// TIA Portal project "SortowanieNiebieskiZielony" (V17)
// Vorlageprojekt für das Buch mit Zielsystem S7-1200

(* hardware
DEVICE "S7-1200-Station_1"  S7-1200 Station
   slot 0: "Baugruppenträger_0"  Rack  V1.0
   slot 1: "PLC_1"  CPU 1211C DC/DC/DC  6ES7 211-1AE40-0XB0  V4.1
*)

// ===== PLC "PLC_1"  CPU 1211C DC/DC/DC =====

VAR_GLOBAL   // PLC tag table "Standard-Variablentabelle"
   "Tag_1" AT %A0.0 : Bool;
   "Tag_2" AT %E0.0 : Bool;
   "Tag_3" AT %E0.1 : Bool;
END_VAR

VAR_GLOBAL   // PLC tag table "Tag table from XML_1"
   "Sensor 1" AT %I6.0 : Bool;
   "Pusher 1 front" AT %I6.1 : Bool;
   "Pusher 1 back" AT %I6.2 : Bool;
   "At pusher 1 exit" AT %I6.3 : Bool;
   "Sensor 2" AT %I6.4 : Bool;
   "Pusher 2 front" AT %I6.5 : Bool;
   "Pusher 2 back" AT %I6.6 : Bool;
   "At pusher 2 exit" AT %I6.7 : Bool;
   "Start" AT %I7.0 : Bool;
   "Reset" AT %I7.1 : Bool;
   "Stop" AT %I7.2 : Bool;
   "Emergency stop" AT %I7.3 : Bool;
   "FACTORY I/O (Running)" AT %I7.4 : Bool;
   "Entry conveyor 1" AT %Q6.0 : Bool;
   "Pusher 1" AT %Q6.1 : Bool;
   "Conveyor 1" AT %Q6.2 : Bool;
   "Entry conveyor 2" AT %Q6.3 : Bool;
   "Pusher 2" AT %Q6.4 : Bool;
   "Conveyor 2" AT %Q6.5 : Bool;
   "Start light" AT %Q6.6 : Bool;
   "Reset light" AT %Q6.7 : Bool;
   "Stop light" AT %Q7.0 : Bool;
   "Vision sensor 1" AT %ID30 : DInt;
   "Vision sensor 2" AT %ID34 : DInt;
   "Counter 1" AT %QD30 : DInt;
   "Counter 2" AT %QD34 : DInt;
END_VAR

// folder: Bloki danych

DATA_BLOCK "DB_FB_SeparationStation"   // DB1
{ S7_Optimized_Access := 'TRUE' }
VERSION : 0.1
// stored: InstanceOfName FB_SeparationStation
"FB_SeparationStation"
BEGIN
END_DATA_BLOCK

// folder: (top level)

ORGANIZATION_BLOCK "Main"   // OB1, LAD, ProgramCycle
TITLE = "Main Program Sweep (Cycle)"
{ S7_Optimized_Access := 'TRUE' }
VERSION : 0.1
   VAR_INPUT
      Initial_Call : Bool;   // Initial call of this OB
      Remanence : Bool;   // =True, if remanent data are available
   END_VAR
BEGIN

REGION Network 1: Konnektierungsbaustein für PLC-Lab
   // Im Netzwerk 1 wird der Konnektierungsbaustein für PLC-Lab aufgerufen.
   // Dieser Aufruf darf nicht entfernt werden!
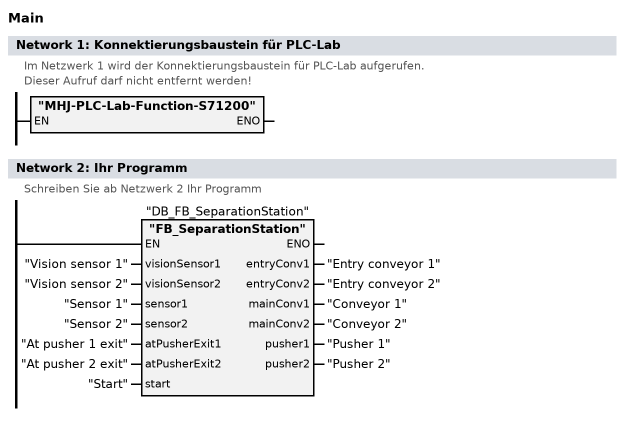
   RUNG wire#powerrail
      "MHJ-PLC-Lab-Function-S71200"()
   END_RUNG
   // the same network as SCL:
   "MHJ-PLC-Lab-Function-S71200"();
END_REGION

REGION Network 2: Ihr Programm
   // Schreiben Sie ab Netzwerk 2 Ihr Programm
   RUNG wire#powerrail
      "DB_FB_SeparationStation"(visionSensor1 := "Vision sensor 1", visionSensor2 := "Vision sensor 2", sensor1 := "Sensor 1", sensor2 := "Sensor 2", atPusherExit1 := "At pusher 1 exit", atPusherExit2 := "At pusher 2 exit", start := "Start", entryConv1 => "Entry conveyor 1", entryConv2 => "Entry conveyor 2", mainConv1 => "Conveyor 1", mainConv2 => "Conveyor 2", pusher1 => "Pusher 1", pusher2 => "Pusher 2")
   END_RUNG
   // the same network as SCL:
   "DB_FB_SeparationStation"(visionSensor1 := "Vision sensor 1",   // "FB_SeparationStation"
                           visionSensor2 := "Vision sensor 2",
                           sensor1 := "Sensor 1",
                           sensor2 := "Sensor 2",
                           atPusherExit1 := "At pusher 1 exit",
                           atPusherExit2 := "At pusher 2 exit",
                           start := "Start",
                           entryConv1 => "Entry conveyor 1",
                           entryConv2 => "Entry conveyor 2",
                           mainConv1 => "Conveyor 1",
                           mainConv2 => "Conveyor 2",
                           pusher1 => "Pusher 1",
                           pusher2 => "Pusher 2");
END_REGION
END_ORGANIZATION_BLOCK

// folder: Funkcje

FUNCTION_BLOCK "FB_SeparationStation"   // FB1, LAD
{ S7_Optimized_Access := 'TRUE' }
VERSION : 0.1
   VAR_INPUT
      visionSensor1 : Int;
      visionSensor2 : Int;
      sensor1 : Bool;
      sensor2 : Bool;
      atPusherExit1 : Bool;
      atPusherExit2 : Bool;
      start : Bool;
   END_VAR
   VAR_OUTPUT
      entryConv1 : Bool;
      entryConv2 : Bool;
      mainConv1 : Bool;
      mainConv2 : Bool;
      pusher1 : Bool;
      pusher2 : Bool;
   END_VAR
   VAR
      cycleStage : Int;
      zbocza : Int;
      colorOfElement : Int;
   END_VAR
   VAR_TEMP   // added for the SCL form of the ladder/FBD networks
      _w1 : Bool;
   END_VAR
BEGIN

REGION Network 1
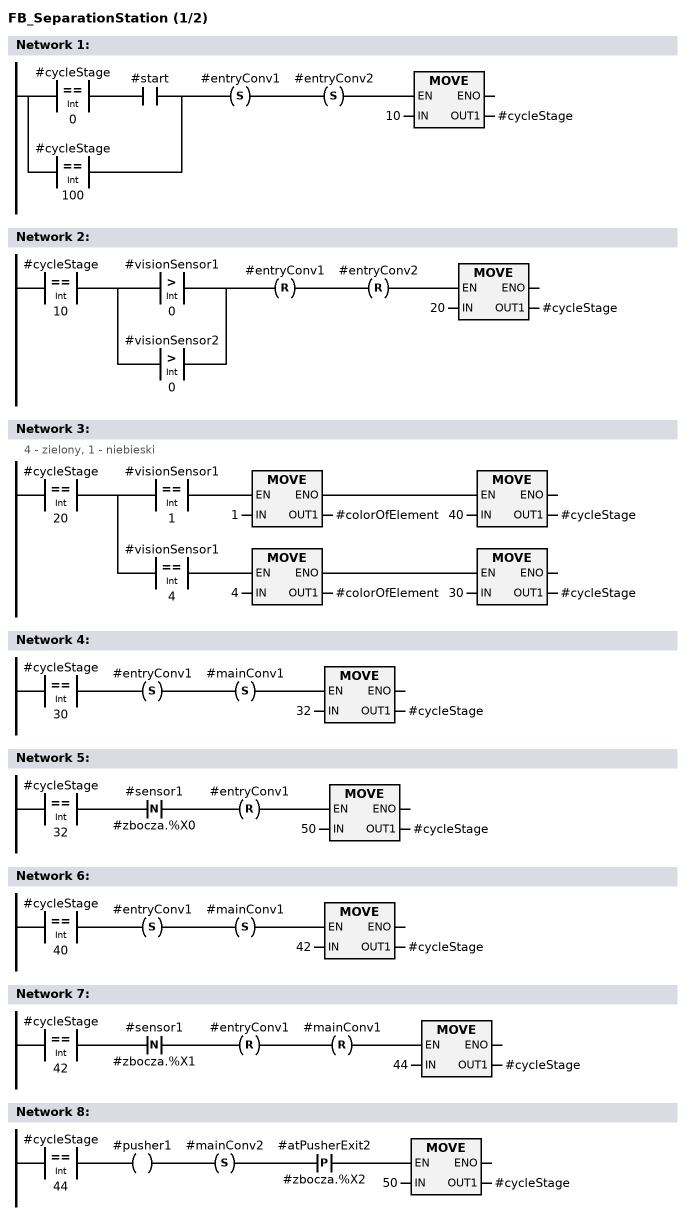
   RUNG wire#powerrail
      { S7_Templates := "SrcType := Int" } EQ_Contact(in1 := #cycleStage, in2 := 0)
      Contact( #start )
      wire#w1
      S_Coil( #entryConv1 )
      S_Coil( #entryConv2 )
      Move(in := 10, out1 => #cycleStage)
   END_RUNG
   RUNG wire#powerrail
      { S7_Templates := "SrcType := Int" } EQ_Contact(in1 := #cycleStage, in2 := 100)
   END_RUNG wire#w1
   // the same network as SCL:
   IF ((#cycleStage = 0) AND #start) OR (#cycleStage = 100) THEN
       #entryConv1 := TRUE;
       #entryConv2 := TRUE;
       #cycleStage := 10;
   END_IF;
END_REGION

REGION Network 2
   RUNG wire#powerrail
      { S7_Templates := "SrcType := Int" } EQ_Contact(in1 := #cycleStage, in2 := 10)
      wire#w1
      { S7_Templates := "SrcType := Int" } GT_Contact(in1 := #visionSensor1, in2 := 0)
      wire#w2
      R_Coil( #entryConv1 )
      R_Coil( #entryConv2 )
      Move(in := 20, out1 => #cycleStage)
   END_RUNG
   RUNG wire#w1
      { S7_Templates := "SrcType := Int" } GT_Contact(in1 := #visionSensor2, in2 := 0)
   END_RUNG wire#w2
   // the same network as SCL:
   IF (#cycleStage = 10) AND ((#visionSensor1 > 0) OR (#visionSensor2 > 0)) THEN
       #entryConv1 := FALSE;
       #entryConv2 := FALSE;
       #cycleStage := 20;
   END_IF;
END_REGION

REGION Network 3
   // 4 - zielony, 1 - niebieski
   RUNG wire#powerrail
      { S7_Templates := "SrcType := Int" } EQ_Contact(in1 := #cycleStage, in2 := 20)
      wire#w1
      { S7_Templates := "SrcType := Int" } EQ_Contact(in1 := #visionSensor1, in2 := 1)
      Move(in := 1, out1 => #colorOfElement)
      Move(in := 40, out1 => #cycleStage)
   END_RUNG
   RUNG wire#w1
      { S7_Templates := "SrcType := Int" } EQ_Contact(in1 := #visionSensor1, in2 := 4)
      Move(in := 4, out1 => #colorOfElement)
      Move(in := 30, out1 => #cycleStage)
   END_RUNG
   // the same network as SCL:
   #_w1 := #cycleStage = 20;
   IF #_w1 AND (#visionSensor1 = 1) THEN
       #colorOfElement := 1;
       #cycleStage := 40;
   END_IF;
   IF #_w1 AND (#visionSensor1 = 4) THEN
       #colorOfElement := 4;
       #cycleStage := 30;
   END_IF;
END_REGION

REGION Network 4
   RUNG wire#powerrail
      { S7_Templates := "SrcType := Int" } EQ_Contact(in1 := #cycleStage, in2 := 30)
      S_Coil( #entryConv1 )
      S_Coil( #mainConv1 )
      Move(in := 32, out1 => #cycleStage)
   END_RUNG
   // the same network as SCL:
   IF #cycleStage = 30 THEN
       #entryConv1 := TRUE;
       #mainConv1 := TRUE;
       #cycleStage := 32;
   END_IF;
END_REGION

REGION Network 5
   RUNG wire#powerrail
      { S7_Templates := "SrcType := Int" } EQ_Contact(in1 := #cycleStage, in2 := 32)
      N_Contact(operand := #sensor1, bit := #zbocza.%X0)
      R_Coil( #entryConv1 )
      Move(in := 50, out1 => #cycleStage)
   END_RUNG
   // the same network as SCL:
   #_w1 := (#cycleStage = 32) AND NOT #sensor1 AND #zbocza.%X0;   // falling edge of #sensor1
   #zbocza.%X0 := #sensor1;
   IF #_w1 THEN
       #entryConv1 := FALSE;
       #cycleStage := 50;
   END_IF;
END_REGION

REGION Network 6
   RUNG wire#powerrail
      { S7_Templates := "SrcType := Int" } EQ_Contact(in1 := #cycleStage, in2 := 40)
      S_Coil( #entryConv1 )
      S_Coil( #mainConv1 )
      Move(in := 42, out1 => #cycleStage)
   END_RUNG
   // the same network as SCL:
   IF #cycleStage = 40 THEN
       #entryConv1 := TRUE;
       #mainConv1 := TRUE;
       #cycleStage := 42;
   END_IF;
END_REGION

REGION Network 7
   RUNG wire#powerrail
      { S7_Templates := "SrcType := Int" } EQ_Contact(in1 := #cycleStage, in2 := 42)
      N_Contact(operand := #sensor1, bit := #zbocza.%X1)
      R_Coil( #entryConv1 )
      R_Coil( #mainConv1 )
      Move(in := 44, out1 => #cycleStage)
   END_RUNG
   // the same network as SCL:
   #_w1 := (#cycleStage = 42) AND NOT #sensor1 AND #zbocza.%X1;   // falling edge of #sensor1
   #zbocza.%X1 := #sensor1;
   IF #_w1 THEN
       #entryConv1 := FALSE;
       #mainConv1 := FALSE;
       #cycleStage := 44;
   END_IF;
END_REGION

REGION Network 8
   RUNG wire#powerrail
      { S7_Templates := "SrcType := Int" } EQ_Contact(in1 := #cycleStage, in2 := 44)
      Coil( #pusher1 )
      S_Coil( #mainConv2 )
      P_Contact(operand := #atPusherExit2, bit := #zbocza.%X2)
      Move(in := 50, out1 => #cycleStage)
   END_RUNG
   // the same network as SCL:
   #pusher1 := #cycleStage = 44;
   IF #pusher1 THEN #mainConv2 := TRUE; END_IF;
   #_w1 := #pusher1 AND #atPusherExit2 AND NOT #zbocza.%X2;   // rising edge of #atPusherExit2
   #zbocza.%X2 := #atPusherExit2;
   IF #_w1 THEN #cycleStage := 50; END_IF;
END_REGION

REGION Network 9
   // 4 - zielony, 1 - niebieski
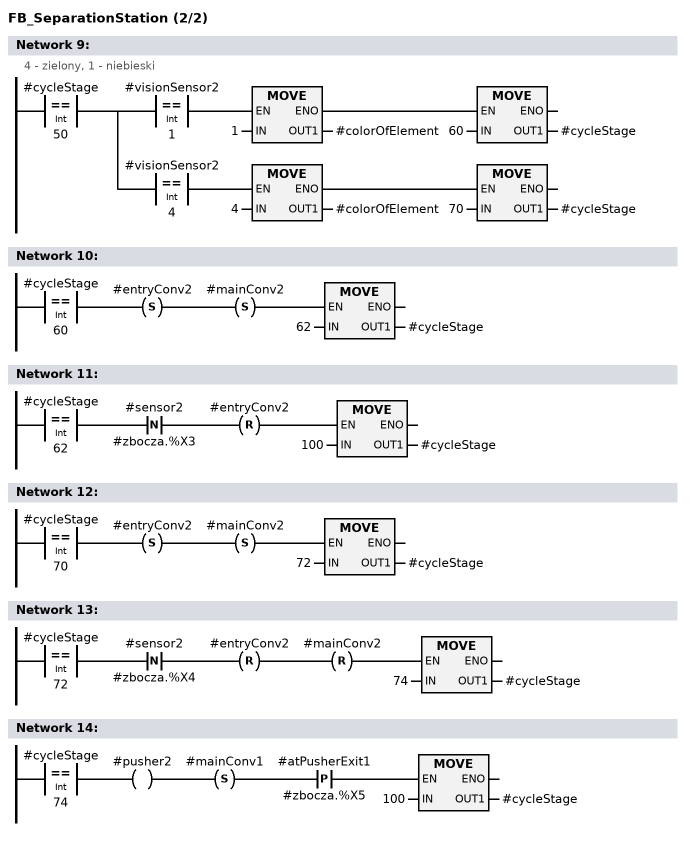
   RUNG wire#powerrail
      { S7_Templates := "SrcType := Int" } EQ_Contact(in1 := #cycleStage, in2 := 50)
      wire#w1
      { S7_Templates := "SrcType := Int" } EQ_Contact(in1 := #visionSensor2, in2 := 1)
      Move(in := 1, out1 => #colorOfElement)
      Move(in := 60, out1 => #cycleStage)
   END_RUNG
   RUNG wire#w1
      { S7_Templates := "SrcType := Int" } EQ_Contact(in1 := #visionSensor2, in2 := 4)
      Move(in := 4, out1 => #colorOfElement)
      Move(in := 70, out1 => #cycleStage)
   END_RUNG
   // the same network as SCL:
   #_w1 := #cycleStage = 50;
   IF #_w1 AND (#visionSensor2 = 1) THEN
       #colorOfElement := 1;
       #cycleStage := 60;
   END_IF;
   IF #_w1 AND (#visionSensor2 = 4) THEN
       #colorOfElement := 4;
       #cycleStage := 70;
   END_IF;
END_REGION

REGION Network 10
   RUNG wire#powerrail
      { S7_Templates := "SrcType := Int" } EQ_Contact(in1 := #cycleStage, in2 := 60)
      S_Coil( #entryConv2 )
      S_Coil( #mainConv2 )
      Move(in := 62, out1 => #cycleStage)
   END_RUNG
   // the same network as SCL:
   IF #cycleStage = 60 THEN
       #entryConv2 := TRUE;
       #mainConv2 := TRUE;
       #cycleStage := 62;
   END_IF;
END_REGION

REGION Network 11
   RUNG wire#powerrail
      { S7_Templates := "SrcType := Int" } EQ_Contact(in1 := #cycleStage, in2 := 62)
      N_Contact(operand := #sensor2, bit := #zbocza.%X3)
      R_Coil( #entryConv2 )
      Move(in := 100, out1 => #cycleStage)
   END_RUNG
   // the same network as SCL:
   #_w1 := (#cycleStage = 62) AND NOT #sensor2 AND #zbocza.%X3;   // falling edge of #sensor2
   #zbocza.%X3 := #sensor2;
   IF #_w1 THEN
       #entryConv2 := FALSE;
       #cycleStage := 100;
   END_IF;
END_REGION

REGION Network 12
   RUNG wire#powerrail
      { S7_Templates := "SrcType := Int" } EQ_Contact(in1 := #cycleStage, in2 := 70)
      S_Coil( #entryConv2 )
      S_Coil( #mainConv2 )
      Move(in := 72, out1 => #cycleStage)
   END_RUNG
   // the same network as SCL:
   IF #cycleStage = 70 THEN
       #entryConv2 := TRUE;
       #mainConv2 := TRUE;
       #cycleStage := 72;
   END_IF;
END_REGION

REGION Network 13
   RUNG wire#powerrail
      { S7_Templates := "SrcType := Int" } EQ_Contact(in1 := #cycleStage, in2 := 72)
      N_Contact(operand := #sensor2, bit := #zbocza.%X4)
      R_Coil( #entryConv2 )
      R_Coil( #mainConv2 )
      Move(in := 74, out1 => #cycleStage)
   END_RUNG
   // the same network as SCL:
   #_w1 := (#cycleStage = 72) AND NOT #sensor2 AND #zbocza.%X4;   // falling edge of #sensor2
   #zbocza.%X4 := #sensor2;
   IF #_w1 THEN
       #entryConv2 := FALSE;
       #mainConv2 := FALSE;
       #cycleStage := 74;
   END_IF;
END_REGION

REGION Network 14
   RUNG wire#powerrail
      { S7_Templates := "SrcType := Int" } EQ_Contact(in1 := #cycleStage, in2 := 74)
      Coil( #pusher2 )
      S_Coil( #mainConv1 )
      P_Contact(operand := #atPusherExit1, bit := #zbocza.%X5)
      Move(in := 100, out1 => #cycleStage)
   END_RUNG
   // the same network as SCL:
   #pusher2 := #cycleStage = 74;
   IF #pusher2 THEN #mainConv1 := TRUE; END_IF;
   #_w1 := #pusher2 AND #atPusherExit1 AND NOT #zbocza.%X5;   // rising edge of #atPusherExit1
   #zbocza.%X5 := #atPusherExit1;
   IF #_w1 THEN #cycleStage := 100; END_IF;
END_REGION
END_FUNCTION_BLOCK

FUNCTION "MHJ-PLC-Lab-Function-S71200" : Void   // FC9000, SCL
{ S7_Optimized_Access := 'TRUE' }
VERSION : 0.1
   VAR_TEMP
      rdTimeReturn : Int;
      outputTime : DTL;
      SyncVal : Byte;
      forVal : Int;
      forVal_2 : Int;
      Value : Byte;
   END_VAR
   VAR CONSTANT
      CompVal : Byte := 16#34;
      Value_01 : Byte := 16#11;
      Value_01_DW : DWord := 16#A165_D992;
      Value_02_DW : DWord := 16#58BE_4401;
   END_VAR
BEGIN

   #Value:=PEEK(area := 16#82,
        dbNumber := 0,
        byteOffset := 511);
   #Value := #Value + 1;

   POKE(area := 16#82,
        dbNumber := 0,
        byteOffset := 511,
        value := #Value);

   POKE(area:=16#81,
        dbNumber:=0,
        byteOffset:=1016,
        value:=#Value_01_DW);
   POKE(area := 16#81,
        dbNumber := 0,
        byteOffset := 1020,
        value := #Value_02_DW);

   POKE(area := 16#81,
        dbNumber := 0,
        byteOffset := 511,
        value := B#16#00);

   FOR #forVal := 0 TO 120 DO
       FOR #forVal_2:=0 TO 10 DO
           #rdTimeReturn:=RD_SYS_T(#outputTime);
           #rdTimeReturn := WR_SYS_T(#outputTime);
           #rdTimeReturn := RD_SYS_T(#outputTime);
           #rdTimeReturn := WR_SYS_T(#outputTime);
       END_FOR;
       #SyncVal:= PEEK(area := 16#81,
                      dbNumber := 0,
                      byteOffset := 511);
       IF #SyncVal = #CompVal THEN
          GOTO M_1;
       END_IF;
   END_FOR;
   RETURN;

   M_1:
   POKE(area := 16#81,
        dbNumber := 0,
        byteOffset := 511,
        value := B#16#0);
END_FUNCTION